Universal Robots PolyScope program: xmlrpc_example.urp

ProgramRoot directory=/programs; kinematics=(a=[0.00016, -0.38186, -0.39231, 0.00004, -0.00003, 0], d=[0.08913, 92.24028, -89.61401, -2.51609, 0.09488, 0.08232], alpha=[1.57018, -0.00203, -0.00723, 1.57069, -1.57067, 0], deltaTheta=[0, -0.45643, 0.40824, 0.04831, -6.28325, -0.00003], status=linearised); lastSavedInVersion=(project__name=Polyscope, major__version=3, minor__version=1, svn__revision=16828, build__date=Jan 26 2015, 14:09:11); name=xmlrpc_example; programVersion=(project__name=Polyscope, major__version=3, minor__version=1, svn__revision=16828, build__date=Jan 26 2015, 14:09:11); robotEnvironmentFileName=default; serialNumberRobot=2014350141
  BeforeStart description=COMMAND_SEQUENCE_BEFORE_PROGRAM_START; name=BeforeStart
    Assignment expr=rpc_factory("xmlrpc","http://172.16.17.1:8080"); operatorValueType=INTEGER; valueSource=EXPRESSION
  MainProgram cartesianAcceleration=1.2; cartesianSpeed=0.25; jointAcceleration=1.3962634015954636; jointSpeed=1.0471975511965976; sharedProcessMoveBlendRadius=0.025; motionType=JOINT_SPACE
    Assignment expr=camera.get_next_pose(ExpressionGeomFeatureNode); operatorValueType=INTEGER; valueSource=EXPRESSION
    Move cartesianAcceleration=1.2; cartesianSpeed=0.25; jointAcceleration=1.3962634015954636; jointSpeed=1.0471975511965976; sharedProcessMoveBlendRadius=0.025; motionType=JOINT_SPACE
      Waypoint blendRadius=0.05; cartesianAcceleration=1.2; cartesianSpeed=0.25; jointAcceleration=1.3962634015954636; jointSpeed=1.0471975511965976; nextMotionTime=2.0; stoppoint=true; useSharedBlendParameter=true; useSharedParameters=true; positionType=VARIABLE_POSITION; name=Waypoint
    Halt 
